PROGRAM MAIN
VAR
	aData		: ARRAY[0..9] OF LREAL := [0, 1, 2, 3, 4, 5, 6, 7, 8, 9];
	fValue		: LREAL;
END_VAR

fValue := F_Calc(ADR(aData), 1, 2);

END_PROGRAM

(* stored: Version 1.1.0.1, ProductVersion 3.1.4022.18
   POU MAIN: Id {7a50fa0f-28bc-47ec-9a4c-1bc085b48504}, SpecialFunc None *)
